% RSLogix 500 project UAS_PLC.RSS, saved by version 8.30.00.16 %
PROJECT "UAS_PLC"    % processor: Bul.1763 MicroLogix 1100 Series B %

PROGRAM FILES
  LAD 2 "MAIN"  4 rungs
  LAD 3 "IO"  10 rungs
  LAD 4 "CONTROL"  6 rungs

DATA FILES
  O0 OUTPUT  5 elements
  I1 INPUT  7 elements
  S2 STATUS  66 elements
  B3 BINARY  1 elements
  T4 TIMER  1 elements
  C5 COUNTER  1 elements
  R6 CONTROL  1 elements
  N7 INTEGER  1 elements
  F8 FLOAT  1 elements

LADDER 2 "MAIN"
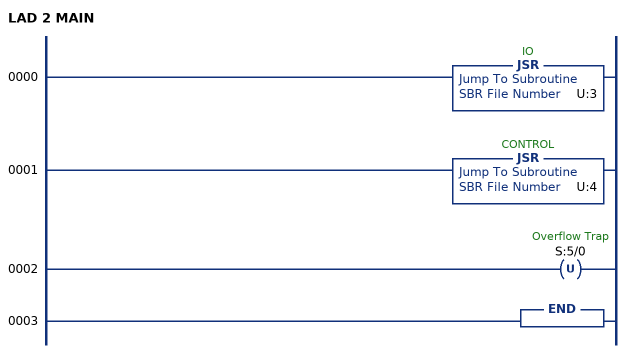
% Rung: 0 %
SOR JSR U:3 EOR
%   U:3  "IO" %
% Rung: 1 %
SOR JSR U:4 EOR
%   U:4  "CONTROL" %
% Rung: 2 %
SOR OTU S:5/0 EOR
%   S:5/0  "Overflow Trap" %
% Rung: 3 %
SOR END EOR

LADDER 3 "IO"
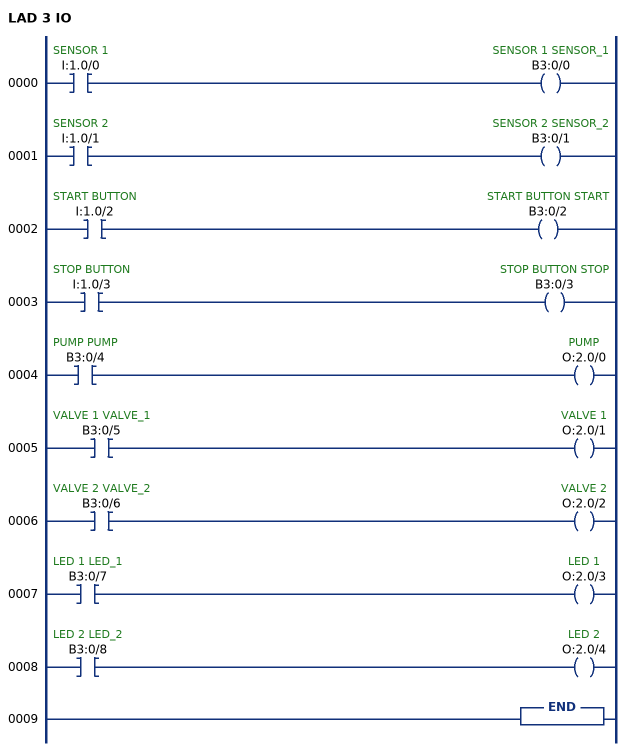
% Rung: 0 %
SOR XIC I:1.0/0 OTE B3:0/0 EOR
%   I:1.0/0  "SENSOR 1" %
%   B3:0/0  SENSOR_1  "SENSOR 1" %
% Rung: 1 %
SOR XIC I:1.0/1 OTE B3:0/1 EOR
%   I:1.0/1  "SENSOR 2" %
%   B3:0/1  SENSOR_2  "SENSOR 2" %
% Rung: 2 %
SOR XIC I:1.0/2 OTE B3:0/2 EOR
%   I:1.0/2  "START BUTTON" %
%   B3:0/2  START  "START BUTTON" %
% Rung: 3 %
SOR XIC I:1.0/3 OTE B3:0/3 EOR
%   I:1.0/3  "STOP BUTTON" %
%   B3:0/3  STOP  "STOP BUTTON" %
% Rung: 4 %
SOR XIC B3:0/4 OTE O:2.0/0 EOR
%   B3:0/4  PUMP  "PUMP" %
%   O:2.0/0  "PUMP" %
% Rung: 5 %
SOR XIC B3:0/5 OTE O:2.0/1 EOR
%   B3:0/5  VALVE_1  "VALVE 1" %
%   O:2.0/1  "VALVE 1" %
% Rung: 6 %
SOR XIC B3:0/6 OTE O:2.0/2 EOR
%   B3:0/6  VALVE_2  "VALVE 2" %
%   O:2.0/2  "VALVE 2" %
% Rung: 7 %
SOR XIC B3:0/7 OTE O:2.0/3 EOR
%   B3:0/7  LED_1  "LED 1" %
%   O:2.0/3  "LED 1" %
% Rung: 8 %
SOR XIC B3:0/8 OTE O:2.0/4 EOR
%   B3:0/8  LED_2  "LED 2" %
%   O:2.0/4  "LED 2" %
% Rung: 9 %
SOR END EOR

LADDER 4 "CONTROL"
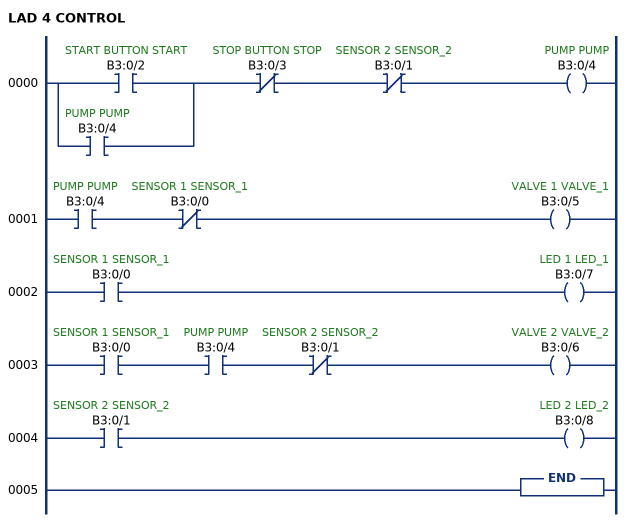
% Rung: 0 %  % edit flag set %
SOR BST XIC B3:0/2 NXB XIC B3:0/4 BND XIO B3:0/3 XIO B3:0/1 OTE B3:0/4 EOR
%   B3:0/2  START  "START BUTTON" %
%   B3:0/4  PUMP  "PUMP" %
%   B3:0/3  STOP  "STOP BUTTON" %
%   B3:0/1  SENSOR_2  "SENSOR 2" %
% Rung: 1 %
SOR XIC B3:0/4 XIO B3:0/0 OTE B3:0/5 EOR
%   B3:0/4  PUMP  "PUMP" %
%   B3:0/0  SENSOR_1  "SENSOR 1" %
%   B3:0/5  VALVE_1  "VALVE 1" %
% Rung: 2 %
SOR XIC B3:0/0 OTE B3:0/7 EOR
%   B3:0/0  SENSOR_1  "SENSOR 1" %
%   B3:0/7  LED_1  "LED 1" %
% Rung: 3 %
SOR XIC B3:0/0 XIC B3:0/4 XIO B3:0/1 OTE B3:0/6 EOR
%   B3:0/0  SENSOR_1  "SENSOR 1" %
%   B3:0/4  PUMP  "PUMP" %
%   B3:0/1  SENSOR_2  "SENSOR 2" %
%   B3:0/6  VALVE_2  "VALVE 2" %
% Rung: 4 %
SOR XIC B3:0/1 OTE B3:0/8 EOR
%   B3:0/1  SENSOR_2  "SENSOR 2" %
%   B3:0/8  LED_2  "LED 2" %
% Rung: 5 %
SOR END EOR
